Omron Sysmac Studio project SPA_P2_V2 (Sysmac Studio 1.23.0.14, StandardProject)

# Controller new_Controller_0: NX1P2-1040DT1 version 1.18
Task PrimaryTask (priority 4, period or condition 2000): Programa0

PROGRAM Programa0
VAR
    analog_input1 : REAL := 0.0;
    out9 : BOOL;
    analog_input2 : REAL;
    out10_1 : BOOL;
    out10_2 : BOOL;
    sensor : REAL;
    analog_input3 : UINT;
    frequency : REAL;
    limit_weight : REAL;
    weight : REAL;
END_VAR

(* Section C9: ladder, written here as Structured Text *)

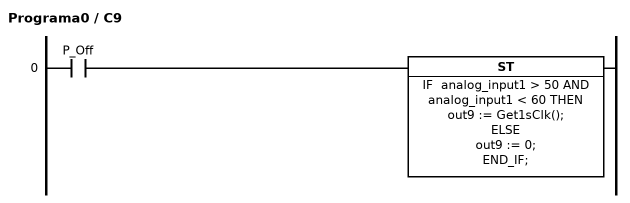
(* Rung 0 *)
IF P_Off THEN
    IF  analog_input1 > 50 AND analog_input1 < 60 THEN
    	out9 := Get1sClk();
    ELSE
    	out9 := 0;
    END_IF;
END_IF;

(* Section C10: ladder, written here as Structured Text *)

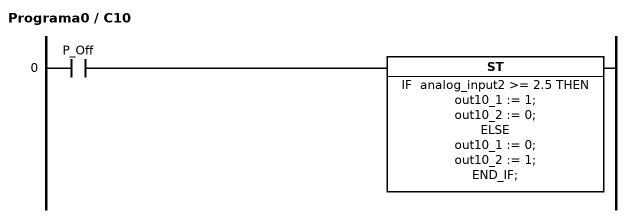
(* Rung 0 *)
IF P_Off THEN
    IF  analog_input2 >= 2.5 THEN
    	out10_1 := 1;
    	out10_2 := 0;
    ELSE
    	out10_1 := 0;
    	out10_2 := 1;
    END_IF;
END_IF;

(* Section C11: ladder, written here as Structured Text *)

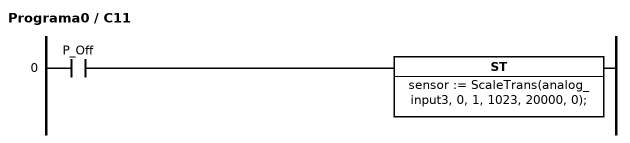
(* Rung 0 *)
IF P_Off THEN
    sensor := ScaleTrans(analog_input3, 0, 1, 1023, 20000, 0);
END_IF;

(* Section C12: ladder, written here as Structured Text *)

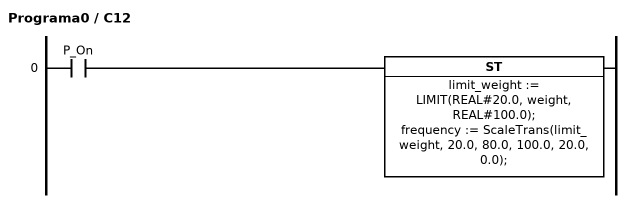
(* Rung 0 *)
IF P_On THEN
    limit_weight := LIMIT(REAL#20.0, weight, REAL#100.0);
    frequency := ScaleTrans(limit_weight, 20.0, 80.0, 100.0, 20.0, 0.0);
END_IF;
END_PROGRAM